// Copies bytes from source to destnation at specified length.
FUNCTION F_MemCpy : POINTER TO BYTE
VAR_INPUT
	pDst,
	pSrc : POINTER TO BYTE;
	Size : T_Size; 
END_VAR
VAR
	i : T_Size := 0;
END_VAR

IF pDst = 0 OR pSrc = 0 OR Size <= 0 THEN RETURN; END_IF
FOR i := 0 TO Size - 1  DO pDst[i] := pSrc[i]; END_FOR
F_MemCpy := pDst;

END_FUNCTION

(* stored: Version 1.1.0.1, ProductVersion 3.1.4024.4
   POU F_MemCpy: Id {ad584eb4-19f4-48bb-b66e-bd11ddf40915}, SpecialFunc None *)
